PROGRAM PRG_BAT_TemperatureControl
VAR
	tempControlMode				: EN_TempControlMode := EN_TempControlMode.TEMP_MODE_MANUAL;  
	
	loopCounter					: DINT := 0;

	(* Controller settings *)
	pwmPeriodinSec			: TIME := T#25S;
	pwmDutyCycle			: REAL := 0.0;	
	pwmOutputValveControl 	: FB_PWM;
	
	//Controling Temperatur for 20°C to 90°C
	CAS_Controller			: FT_PID_CAS;
	
	//Controling Temperatur above 90°C
	STERI_Controller		: FT_PID_STERI;
	
	//GET_GAINS
	GET_GAINS				: FT_GET_GAINS;
	//GAINS JACKET
	kp_J					: REAL ;
	ki_J					: REAL ;
	//GAINS CELL
	kp_C					: REAL ;
	ki_C					: REAL ;
	kd_C					: REAL ;
	
	//Traking time - anti-windup 
	tr_J					: REAL := 1.0;
	tr_C					: REAL := 1.0;
	//is used for changing the status from heating <-> cooling 
	TargetTemp_old 			: REAL ;
	
	// Cooling or Heating for MODE_HEATCOOL;
	COOLING 				: BOOL := FALSE;
	HEATING					: BOOL := FALSE;
	CHANGE_TO_HEATING		: BOOL := FALSE;	
	
	errorTemp				: REAL := 0.0;
	pidReset				: BOOL := FALSE;
		
	evtSteriStart			: DetectEvent;
	evtSteriStop			: DetectEvent;
		
	evtTempControlStart		: DetectEvent;
	evtTempControlStop		: DetectEvent;
	
	windUpResetTimer		: TON;
	windUpResetTime			: TIME := T#30S;
	
	maxValveOnTimer		 	: TON;
	maxValveOnTime			: TIME := T#25S;	
	
	evtPidReset				: DetectEvent;
END_VAR

(* jacket temperature input *)
jacketTempC := INT_TO_REAL(jacketTempRaw)/32768.0*200.0 -50.0;
jacketTempK := jacketTempC + 273.15;
tOrpCurrent;
tPhCurrent;
currentMeanTemp;


evtSteriStart(		newSignalValue := steriStart);
evtSteriStop(		newSignalValue := steriStop);
evtTempControlStart(newSignalValue := tempControlStart);
evtTempControlStop(	newSignalValue := tempControlStop);
evtPidReset( 		newSignalValue := pidReset);


IF evtSteriStart.eventDetected = TASTEVT_PositiveEdge THEN
	steriStart := FALSE;
	pumpOn := FALSE;
	CAS_Controller( RST:= TRUE );
	STERI_Controller(RST:=TRUE);
	tempControlMode	:= EN_TempControlMode.TEMP_MODE_STERI;
	tempControlRunning := FALSE;
	steriRunning := TRUE;
	steriValve := FALSE;
	coldValve := FALSE;
	hotValve := FALSE;
	(* Set remaining steri temp *)
	remainingSteriTimeInMs := targetSteriTimeMinutes*60*1000; 
END_IF

IF evtTempControlStart.eventDetected = TASTEVT_PositiveEdge THEN
	tempControlStart := FALSE;
	pumpOn := FALSE;
	CAS_Controller( RST:= TRUE );
	STERI_Controller(RST:=TRUE);
	tempControlMode	:= EN_TempControlMode.TEMP_MODE_HEATCOOL;
	tempControlRunning := TRUE;
	steriRunning := FALSE;
	steriValve := FALSE;
	coldValve := FALSE;
	hotValve := FALSE;
END_IF

IF 	evtSteriStop.eventDetected = TASTEVT_PositiveEdge OR
 	evtTempControlStop.eventDetected = TASTEVT_PositiveEdge 
THEN
	steriStop := FALSE;
	tempControlStop := FALSE;
	pumpOn := FALSE;
	CAS_Controller( RST:= TRUE );
	STERI_Controller(RST:=TRUE);
	tempControlRunning := FALSE;
	steriRunning := FALSE;
	tempControlMode	:= EN_TempControlMode.TEMP_MODE_MANUAL;
	coldValve := FALSE;
	hotValve := FALSE;
	steriValve := FALSE;
	(* TODO: Reset Steri Timer *)
END_IF

(* check if current temperature reading actually valid, otherwise stop any type of temperature control *)

IF NOT currentTempValid THEN
	tempControlMode := EN_TempControlMode.TEMP_MODE_MANUAL;
END_IF


CASE tempControlMode OF
	EN_TempControlMode.TEMP_MODE_MANUAL:
		pumpOn := FALSE;
		CAS_Controller( RST:= TRUE );
		STERI_Controller(RST:=TRUE);
		coldValve := FALSE;
		hotValve := FALSE;
		steriValve := FALSE;
		
		
	EN_TempControlMode.TEMP_MODE_HEATCOOL:
		
		pumpOn := TRUE;
		(* errorTemp := targetControlTemp - currentMeanTemp; *)
		errorTemp := FUN_ComputeMovingSetPoint(currentTemp := currentMeanTemp, targetSetPoint := targetControlTemp) - currentMeanTemp;
		
		//If temperature close to targetTemp - change to heating
		IF COOLING = TRUE THEN
			IF (errorTemp<2) THEN
				CHANGE_TO_HEATING := TRUE;
			ELSE
				CHANGE_TO_HEATING := FALSE;			
			END_IF
		END_IF
		
		//Setting Heating or Cooling only when TargetTemp is changed or ...
		// 	...	errorTemp is lower than 2 Degree so it changes to heating - has to be adjusted
		IF (TargetTemp_old = targetControlTemp) AND (CHANGE_TO_HEATING = FALSE) THEN
			;
			ELSE
				//-----COOLING-----
			IF (TargetTemp_old > targetControlTemp) AND (targetControlTemp <40) THEN
				COOLING := TRUE;
				HEATING := FALSE;
				GET_GAINS( 	TEMP := targetControlTemp,
							MODE := 0,);
				kp_J := GET_GAINS.K_P_J;
				ki_J := GET_GAINS.K_I_J;
				tr_J := GET_GAINS.T_R_J;
 				kp_C := GET_GAINS.K_P_C;
				ki_C := GET_GAINS.K_I_C;
				kd_C := GET_GAINS.K_D_C;
				tr_C := GET_GAINS.T_R_C;
				//-----HEATING-----
			ELSE
				COOLING := FALSE;
				HEATING := TRUE;	
				GET_GAINS( 	TEMP := targetControlTemp,
							MODE := 1,);
				kp_J := GET_GAINS.K_P_J;
				ki_J := GET_GAINS.K_I_J;
				tr_J := GET_GAINS.T_R_J;
 				kp_C := GET_GAINS.K_P_C;
				ki_C := GET_GAINS.K_I_C;
				kd_C := GET_GAINS.K_D_C;
				tr_C := GET_GAINS.T_R_C;
			END_IF
		END_IF
		//Save old TargetTemp
		TargetTemp_old := TargetControlTemp;	 
		
		//Start Temp. Controller
		CAS_Controller(	T_ERR_C := errorTemp,		//Cell Temperatur error 
						K_P_J 	:= kp_J,
						K_I_J 	:= ki_J,
						T_R_J 	:= tr_J,			//Tracking time used for Anti-Wind up
						K_P_C 	:= kp_C,	
						K_I_C 	:= ki_C,
						K_D_C 	:= kd_C,			
						T_R_C	:= tr_C, 			//Tracking time used for Anti-Wind up
						LIM_L 	:= 0.0,				//Min. Temp for Jacket
						LIM_H 	:= 90.0,			//Max. Temp for Jacket
						RST 	:= pidReset,
						);
												
		pwmDutyCycle := CAS_Controller.P_J_Controll.Y; (* !! pwm block cannot handle negative inputs *)
		//pwmDutyCycle := 1;

		pwmOutputValveControl(pwmCycleTime:=pwmPeriodinSec, pwmDutyCycle:=pwmDutyCycle);	
						
		IF  HEATING = TRUE THEN			 	//heating 
			coldValve := FALSE;
			hotValve := pwmOutputValveControl.Q;
			steriValve := FALSE;
			
		ELSIF COOLING = TRUE THEN			//cooling 
			coldValve := pwmOutputValveControl.Q;
			hotValve := FALSE;
			steriValve := FALSE;
			
		ELSE								//ERROR STATE?
			coldValve := FALSE;
			hotValve := FALSE;
			steriValve := FALSE;
		END_IF
		
//----------------------------------------------STERIL-------------------------------------------------------------------			
	EN_TempControlMode.TEMP_MODE_STERI:
		pumpOn := FALSE;
		errorTemp := targetSteriTemp - currentMeanTemp;
		
		//Setting Heating or Cooling only when TargetTemp is changed
		IF TargetTemp_old = targetControlTemp THEN
			;
			ELSE
			IF (TargetTemp_old > targetControlTemp) THEN
				COOLING := FALSE;
				HEATING := FALSE;

			ELSE
				COOLING := FALSE;
				HEATING := TRUE;	
				GET_GAINS( 	TEMP := targetControlTemp,
							MODE := 1,);
				kp_C := GET_GAINS.K_P_C;
				ki_C := GET_GAINS.K_I_C;
				kd_C := GET_GAINS.K_D_C;
				tr_C := GET_GAINS.T_R_C;
			END_IF
		END_IF
		//Save old TargetTemp
		TargetTemp_old := TargetControlTemp;	
		//Start Temp. Controller
		STERI_Controller(	
						T_ERR_C := errorTemp,		//Cell Temperatur error 
						K_P_C 	:= kp_C,	
						K_I_C 	:= ki_C,
						K_D_C 	:= kd_C,			
						T_R_C	:= tr_C, 			//Tracking time used for Anti-Wind up
						LIM_L 	:= 0.0,				//Min. Temp for Jacket
						LIM_H 	:= 1.0,				//Max. Temp for Jacket
						RST 	:= pidReset,
						);
						
		pwmDutyCycle := STERI_Controller.Y; 	
		//pwmDutyCycle := 0.5;
		
		pwmOutputValveControl(pwmCycleTime:=pwmPeriodinSec, pwmDutyCycle:=pwmDutyCycle);
				
		IF HEATING = TRUE THEN
			(* heating *)
			coldValve 	:= FALSE;
			steriValve 	:= pwmOutputValveControl.Q;
			hotValve 	:= FALSE;
			
		ELSE
			(* cooling *)
			steriValve 	:= FALSE;
			hotValve 	:= FALSE;			
		END_IF
		
		IF currentMeanTemp > (targetSteriTemp-0.5) THEN
			(* count down 10 ms each cycle *)
			remainingSteriTimeInMs := remainingSteriTimeInMs - 10;
			IF remainingSteriTimeInMs < 0 THEN
				tempControlMode := EN_TempControlMode.TEMP_MODE_MANUAL;
				steriValve := FALSE;
				coldValve := FALSE;
				steriStop := TRUE;
			END_IF
		END_IF		
		remainingSteriTimeMinutes := DINT_TO_REAL(remainingSteriTimeInMs)/(60.0*1000.0);
	
	
END_CASE
 
IF evtPidReset.eventDetected = TASTEVT_PositiveEdge THEN
	pidReset := FALSE;
	CAS_Controller(RST:=TRUE);
	STERI_Controller(RST:=TRUE);
	pidResetCounter := pidResetCounter + 1;
	steriValve := FALSE;
	coldValve := FALSE;
	hotValve := FALSE;
END_IF

END_PROGRAM

(* stored: Version 1.1.0.1, ProductVersion 3.1.4022.12
   POU PRG_BAT_TemperatureControl: Id {bda1fa6f-ddc5-471e-a247-4df659a0e1df}, SpecialFunc None *)
